// TIA Portal V20 export
FUNCTION_BLOCK "FB_LoaderMain"   // FB203, SCL
{ S7_Optimized_Access := 'TRUE' }
// stored: AutoNumber false, MemoryReserve 100, SetENOAutomatically false
   VAR
      sSynchroMode : Bool;
      sSynchroPosition : Bool;
      sLoaderStartRequest : Bool;
      sTimeMeasure : "FB_TimeMeasure";
      sRT_LoaderStartRequest { S7_SetPoint := 'True'} : R_TRIG;
      sBwConsecutiveCtrl { S7_SetPoint := 'True'} : "FB_Consecutive";
      sRT_ConsecutiveCtrl { S7_SetPoint := 'True'} : R_TRIG;
   END_VAR
BEGIN
   REGION Description header 
       //==================================================================================
       // POSALUX Swiss SA / (C) Copyright 2025
       //----------------------------------------------------------------------------------
       // Title: 
       // Comment/Function: 
       // Author: Fabien WALDT
       // Engineering: TIA Portal v17
       //----------------------------------------------------------------------------------
       // Change log table:
       // Version  | Date     | Expert in charge | Changes applied
       // ---------|----------|------------------|-----------------------------------------
       // 00.00.01 | 20251013 | WFA              | First released version
       // =================================================================================
   END_REGION

   REGION Options
       // Ext Load Unload
       "DB_LoaderOptions".ExtLoadUnload.SeparatePos := FALSE;
       "DB_LoaderOptions".ExtLoadUnload.CommonPos := TRUE;
       // Part Control
       "DB_LoaderOptions".PartControl.Individual := FALSE;
       "DB_LoaderOptions".PartControl.Common := TRUE;
       "DB_LoaderOptions".PartControl.Disabled := FALSE;
       "DB_LoaderOptions".PartControl.AnalogMeasure := FALSE;
       "DB_LoaderOptions".PartControl.DigitalMeasure := TRUE;
       // BW Load Unload
       "DB_LoaderOptions".BwLoadUnload.SeparatePos := TRUE;
       "DB_LoaderOptions".BwLoadUnload.CommonPos := FALSE;
       // BW Control
       "DB_LoaderOptions".BwControl.UndrilledDrilledCtrlSeparate := TRUE;
       "DB_LoaderOptions".BwControl.UndrilledDrilledCtrlCommon := FALSE;
       "DB_LoaderOptions".BwControl.Disabled := FALSE;
       // Int Load Unload
       "DB_LoaderOptions".IntLoadUnload.SeparatePos := FALSE;
       "DB_LoaderOptions".IntLoadUnload.CommonPos := TRUE;
   END_REGION

   REGION History Activation
       // Shuttle 1
       "DB_LoaderShuttle1".sMain.sHistory.Activation := TRUE;
       "DB_LoaderShuttle1".sShuttleInt.sHistory.Activation := TRUE;
       "DB_LoaderShuttle1".sShuttleExt.sHistory.Activation := TRUE;
       "DB_LoaderShuttle1".sControlIn.sHistory.Activation := TRUE;
       "DB_LoaderShuttle1".sControlOut.sHistory.Activation := TRUE;
       "DB_LoaderShuttle1".sIntLoadUnload.sHistory.Activation := TRUE;
       "DB_LoaderShuttle1".sIntLoadUnloadOP.sHistory.Activation := TRUE;
       "DB_LoaderShuttle1".sExtLoadUnload.sHistory.Activation := TRUE;
       "DB_LoaderShuttle1".sBwLoadUnload.sHistory.Activation := TRUE;
       "DB_LoaderShuttle1".sBwControlIn.sHistory.Activation := TRUE;
       "DB_LoaderShuttle1".sActBwControlIn.sHistory.Activation := TRUE;
       "DB_LoaderShuttle1".sActPartControlIn.sHistory.Activation := TRUE;
       "DB_LoaderShuttle1".sActPartControlOut.sHistory.Activation := TRUE;
       "DB_LoaderShuttle1".sBlowing.sHistory.Activation := TRUE;

       // Shuttle 2
       "DB_LoaderShuttle2".sMain.sHistory.Activation := TRUE;
       "DB_LoaderShuttle2".sShuttleInt.sHistory.Activation := TRUE;
       "DB_LoaderShuttle2".sShuttleExt.sHistory.Activation := TRUE;
       "DB_LoaderShuttle2".sControlIn.sHistory.Activation := TRUE;
       "DB_LoaderShuttle2".sControlOut.sHistory.Activation := TRUE;
       "DB_LoaderShuttle2".sIntLoadUnload.sHistory.Activation := TRUE;
       "DB_LoaderShuttle2".sIntLoadUnloadOP.sHistory.Activation := TRUE;
       "DB_LoaderShuttle2".sExtLoadUnload.sHistory.Activation := TRUE;
       "DB_LoaderShuttle2".sBwLoadUnload.sHistory.Activation := TRUE;
       "DB_LoaderShuttle2".sBwControlIn.sHistory.Activation := TRUE;
       "DB_LoaderShuttle2".sActBwControlIn.sHistory.Activation := TRUE;
       "DB_LoaderShuttle2".sActPartControlIn.sHistory.Activation := TRUE;
       "DB_LoaderShuttle2".sActPartControlout.sHistory.Activation := TRUE;
       "DB_LoaderShuttle2".sBlowing.sHistory.Activation := TRUE;
   END_REGION

   REGION Loader Start
       IF "LBP_Chan1".MDyn[75] AND ("DB_WorkingModes".sAuto OR "DB_WorkingModes".sSemiAuto) THEN
           #sLoaderStartRequest := TRUE;
       ELSIF
           ("DB_WorkingModes".sEmptying AND "DB_PartManagement".sPosition.sMachineEmpty)
          OR NOT "DB_PowerOn".sMachineReadySoft
          OR  "MCP1_In".reset THEN
           #sLoaderStartRequest := FALSE;
       END_IF;

           #sRT_LoaderStartRequest(CLK := #sLoaderStartRequest);
           IF NOT "LBP_ModeGroup".E_JOG AND #sRT_LoaderStartRequest.Q THEN
               IF "DB_HMISetting".Shuttle1Enable THEN
                   "DB_LoaderShuttle1".sMain.iJobReq := TRUE;
               END_IF;
               IF "DB_HMISetting".Shuttle2Enable THEN
                   "DB_LoaderShuttle2".sMain.iJobReq := TRUE;
               END_IF;
           ELSIF NOT #sLoaderStartRequest THEN
               "DB_LoaderShuttle1".sMain.iJobReq := FALSE;
               "DB_LoaderShuttle2".sMain.iJobReq := FALSE;
           END_IF;
   END_REGION

   REGION Shuttle 1
       "DB_LoaderShuttle1"(iGripperReserved := "DB_GestionGripper".sGripperStatus.DrivedByShuttle1,
                           iGripperReleased := NOT "DB_GestionGripper".sGripperStatus.DrivedByShuttle1,
                           iShuttleMoving := "DB_LoaderAxis".sU1Positioning,
                           iShuttleInPos := "DB_LoaderAxis".sU1InPos,
                           iAxisV_Moving := "DB_LoaderAxis".sVPositioning,
                           iAxisV_InPos := "DB_LoaderAxis".sVInPos,
                           iAxisW_Moving := "DB_LoaderAxis".sWPositioning,
                           iAxisW_InPos := "DB_LoaderAxis".sWInPos,
                           oExtGateOpenReq => "DB_LoaderShuttle1".oExtGateOpenReq,
                           oExtGateCloseReq => "DB_LoaderShuttle1".oExtGateCloseReq,
                           oIntGateOpenReq => "DB_LoaderShuttle1".oIntGateOpenReq,
                           oIntGateCloseReq => "DB_LoaderShuttle1".oIntGateCloseReq,
                           oLoadGripperCloseReq => "DB_LoaderShuttle1".oLoadGripperCloseReq,
                           oUnloadGripperOpenReq => "DB_LoaderShuttle1".oUnloadGripperOpenReq,
                           oShuttleStartReq => "DB_LoaderShuttle1".oShuttleStartReq,
                           oShuttlePosSetPoint => "DB_LoaderAxis".iU1PosSetPoint,
                           oAxisVStartReq => "DB_LoaderShuttle1".oAxisVStartReq,
                           oAxisVPosSetPoint => "DB_LoaderShuttle1".oAxisVPosSetPoint,
                           oAxisWStartReq => "DB_LoaderShuttle1".oAxisWStartReq,
                           oAxisWPosSetPoint => "DB_LoaderShuttle1".oAxisWPosSetPoint);
   END_REGION

   REGION Shuttle 2
       "DB_LoaderShuttle2"(iGripperReserved := "DB_GestionGripper".sGripperStatus.DrivedByShuttle2,
                           iGripperReleased :=  NOT "DB_GestionGripper".sGripperStatus.DrivedByShuttle2,
                           iShuttleMoving := "DB_LoaderAxis".sU2Positioning,
                           iShuttleInPos := "DB_LoaderAxis".sU2InPos,
                           iAxisV_Moving := "DB_LoaderAxis".sVPositioning,
                           iAxisV_InPos := "DB_LoaderAxis".sVInPos,
                           iAxisW_Moving := "DB_LoaderAxis".sWPositioning,
                           iAxisW_InPos := "DB_LoaderAxis".sWInPos,
                           oExtGateOpenReq => "DB_LoaderShuttle2".oExtGateOpenReq,
                           oExtGateCloseReq => "DB_LoaderShuttle2".oExtGateCloseReq,
                           oIntGateOpenReq => "DB_LoaderShuttle2".oIntGateOpenReq,
                           oIntGateCloseReq => "DB_LoaderShuttle2".oIntGateCloseReq,
                           oLoadGripperCloseReq => "DB_LoaderShuttle2".oLoadGripperCloseReq,
                           oUnloadGripperOpenReq => "DB_LoaderShuttle2".oUnloadGripperOpenReq,
                           oShuttleStartReq => "DB_LoaderShuttle2".oShuttleStartReq,
                           oShuttlePosSetPoint => "DB_LoaderAxis".iU2PosSetPoint,
                           oAxisVStartReq => "DB_LoaderShuttle2".oAxisVStartReq,
                           oAxisVPosSetPoint => "DB_LoaderShuttle2".oAxisVPosSetPoint,
                           oAxisWStartReq => "DB_LoaderShuttle2".oAxisWStartReq,
                           oAxisWPosSetPoint => "DB_LoaderShuttle2".oAxisWPosSetPoint);
   END_REGION

   REGION Loader Axis
       IF "DB_LoaderShuttle1".oAxisVStartReq THEN
           "DB_LoaderAxis".iVPosSetPoint := "DB_LoaderShuttle1".oAxisVPosSetPoint;
       ELSIF "DB_LoaderShuttle2".oAxisVStartReq THEN
           "DB_LoaderAxis".iVPosSetPoint := "DB_LoaderShuttle2".oAxisVPosSetPoint;
       ELSIF "DB_LoaderFixture".oAxisV_StartReq THEN
           "DB_LoaderAxis".iVPosSetPoint := "DB_LoaderFixture".oAxisV_PosSetPoint;
       END_IF;

       IF "DB_LoaderShuttle1".oAxisWStartReq THEN
           "DB_LoaderAxis".iWPosSetPoint := "DB_LoaderShuttle1".oAxisWPosSetPoint;
       ELSIF "DB_LoaderShuttle2".oAxisWStartReq THEN
           "DB_LoaderAxis".iWPosSetPoint := "DB_LoaderShuttle2".oAxisWPosSetPoint;
       ELSIF "DB_LoaderFixture".oAxisW_StartReq THEN
           "DB_LoaderAxis".iWPosSetPoint := "DB_LoaderFixture".oAxisW_PosSetPoint;
       END_IF;

       // Demande Axes gérés par PLC (/Mode Jog)
       IF "LBP_ModeGroup".E_MDA OR "LBP_ModeGroup".E_AUTO THEN
           "DB_LoaderAxis".iPLCModeReq := TRUE;
       ELSE
           "DB_LoaderAxis".iPLCModeReq := FALSE;
       END_IF;

       // Demande Axes gérés par NC (Mode Jog)
       // Jog Mode OR R_Trig Auto Mode
           IF "LBP_ModeGroup".E_JOG  THEN
           "DB_LoaderAxis".iCNCModeReq := TRUE;
       ELSE
           "DB_LoaderAxis".iCNCModeReq := FALSE;
       END_IF;

       "DB_LoaderAxis"(iPLCModeReq := "DB_LoaderAxis".iPLCModeReq,
                       iCNCModeReq := "DB_LoaderAxis".iCNCModeReq,
                       iU1StartReq := "DB_LoaderShuttle1".oShuttleStartReq,
                       iU2StartReq := "DB_LoaderShuttle2".oShuttleStartReq,
                       iVStartReq := "DB_LoaderShuttle1".oAxisVStartReq OR "DB_LoaderShuttle2".oAxisVStartReq OR "DB_LoaderFixture".oAxisV_StartReq,
                       iWStartReq := "DB_LoaderShuttle1".oAxisWStartReq OR "DB_LoaderShuttle2".oAxisWStartReq OR "DB_LoaderFixture".oAxisW_StartReq,
                       iU1PosSetPoint := "DB_LoaderAxis".iU1PosSetPoint,
                       iU2PosSetPoint := "DB_LoaderAxis".iU2PosSetPoint,
                       iVPosSetPoint := "DB_LoaderAxis".iVPosSetPoint,
                       iWPosSetPoint := "DB_LoaderAxis".iWPosSetPoint,
                       oU1InPos => "DB_LoaderAxis".oU1InPos,
                       oU2InPos => "DB_LoaderAxis".oU2InPos,
                       oVInPos => "DB_LoaderAxis".oVInPos,
                       oWInPos => "DB_LoaderAxis".oWInPos);
   END_REGION

   REGION Safety Gate
       "DB_GestionSafetyGate"();
   END_REGION

   REGION Gripper
       "DB_GestionGripper"();
   END_REGION

   REGION Fixture
       "DB_GestionFixture"();
   END_REGION

   REGION Syncro Mode 
       // WFA Tester le cycle en supprimant cette REGION (voir tSynchroMode dans FB_GestionSafetyGate)
       #sSynchroMode := "DB_LoaderShuttle1".sMain.sInterface.SequenceRun
       AND "DB_LoaderShuttle2".sMain.sInterface.SequenceRun
       AND (("DB_LoaderShuttle1".sShuttleInt.oExtGateOpenReq AND "DB_LoaderShuttle2".sShuttlePosSas)
       OR ("DB_LoaderShuttle1".sShuttleInt.oIntGateOpenReq AND "DB_LoaderShuttle2".sShuttlePosInt)
       OR ("DB_LoaderShuttle1".sShuttleExt.oExtGateOpenReq AND "DB_LoaderShuttle2".sShuttlePosExt)
       OR ("DB_LoaderShuttle1".sShuttleExt.oIntGateOpenReq AND "DB_LoaderShuttle2".sShuttlePosSas)
       OR ("DB_LoaderShuttle2".sShuttleInt.oExtGateOpenReq AND "DB_LoaderShuttle1".sShuttlePosSas)
       OR ("DB_LoaderShuttle2".sShuttleInt.oIntGateOpenReq AND "DB_LoaderShuttle1".sShuttlePosInt)
       OR ("DB_LoaderShuttle2".sShuttleExt.oExtGateOpenReq AND "DB_LoaderShuttle1".sShuttlePosExt)
       OR ("DB_LoaderShuttle2".sShuttleExt.oIntGateOpenReq AND "DB_LoaderShuttle1".sShuttlePosSas));
   END_REGION

   REGION Time Measure
       #sTimeMeasure(iImpulsion := "DB_GestionGripper".sLoadGripperCloseReq,
                     iPLC_DateAndTime := "DB_ReadDateAndTime".sDateAndTime);
   END_REGION

   REGION Consecutive
       IF "DB_OPC_Machine".Parameters.ConsecutiveBwIn > 0 THEN
           #sBwConsecutiveCtrl(iReset := #sBwConsecutiveCtrl.oConsecutiveError AND ("DB_McpKeyboardSignals".sAlarmReset.sKeySWStatus OR "MCP1_In".reset),
                               iGoodEntry := "DB_LoaderShuttle1".sBwControlIn.oBwControlOK OR "DB_LoaderShuttle2".sBwControlIn.oBwControlOK,
                               iBadEntry := "DB_LoaderShuttle1".sBwControlIn.oBwControlNOK OR "DB_LoaderShuttle2".sBwControlIn.oBwControlNOK,
                               iPresetValue := "DB_OPC_Machine".Parameters.ConsecutiveBwIn,
                               oConsecutiveError => #sBwConsecutiveCtrl.oConsecutiveError);

           #sRT_ConsecutiveCtrl(CLK := #sBwConsecutiveCtrl.oConsecutiveError);
           IF #sRT_ConsecutiveCtrl.Q THEN
               "LBP_AlarmMsgs".UserA[03].A70UUxx[27] := TRUE;
           END_IF;
       END_IF;
   END_REGION
END_FUNCTION_BLOCK
